{attribute 'qualified_only'}
VAR_GLOBAL
	Logger			: FB_Logger;
	ADSNetID_CAN	: STRING(23) := '5.156.6.243.3.1';	// ADSNETID of the CAN module
	NodeID			: BYTE :=2;								// Node ID of the controller	
END_VAR

(* stored: Version 1.1.0.1, ProductVersion 3.1.4024.11
   GVL GLB: Id {7cf4333b-9e18-4f76-aafc-2f9adaa22408} *)
